FUNCTION_BLOCK PLCopenCommand IMPLEMENTS IPLCopenCommand
VAR
    _PLCopenCommand : PLCopenCommandInternal;
END_VAR

// Copyright (c) 2024 Loupe (https://loupe.team), provided under the MIT License.

IF _PLCopenCommand._status <> PLCopenStatusBase.BUSY AND NOT Execute THEN
    _PLCopenCommand._status := PLCopenStatusBase.NOT_ENABLED;
END_IF

METHOD Aborted : BOOL
VAR_INPUT
END_VAR
// Copyright (c) 2024 Loupe (https://loupe.team), provided under the MIT License.

_PLCopenCommand._status := PLCopenStatusBase.ABORTED;

Remote.Aborted();
Remote := 0;
END_METHOD

METHOD AbortPreviousCommands : BOOL
VAR_INPUT
    newCommand : IPLCopenCommand;
END_VAR
VAR
    i : USINT;
END_VAR
// Copyright (c) 2024 Loupe (https://loupe.team), provided under the MIT License.

//If there is a remote, abort it here
//Don't use this^.abort() because we don't want about ourselves
Remote.Aborted();
Remote := 0;

//Abort any related commands
FOR i := 0 TO GVLTcCommando.MAX_RELATED_GROUPS DO
    IF _PLCopenCommand._commandGroups[i] <> 0 THEN
        _PLCopenCommand._commandGroups[i].AbortPreviousCommands(newCommand);
    END_IF
END_FOR
END_METHOD

METHOD FINAL BaseSize : ULINT
// Copyright (c) 2024 Loupe (https://loupe.team), provided under the MIT License.

BaseSize := SIZEOF(THIS^);
END_METHOD

PROPERTY Consume : BOOL
GET
// Copyright (c) 2024 Loupe (https://loupe.team), provided under the MIT License.

Consume := _PLCopenCommand._Execute;

IF _PLCopenCommand._Execute THEN
    //	THIS^.AbortPreviousCommands( THIS^ );//This is meant to abort if the command comes locally
    _PLCopenCommand._status := PLCopenStatusBase.BUSY;
END_IF

_PLCopenCommand._Execute := FALSE;
END_GET
END_PROPERTY

METHOD Errored : BOOL
VAR_INPUT
    ID : INT;
END_VAR
// Copyright (c) 2024 Loupe (https://loupe.team), provided under the MIT License.

CASE ID OF
    //Any of these statuses are invalid to return as an error.
    //Override to error
    PLCopenStatusBase.BUSY,
        PLCopenStatusBase.ENABLED_WAITING,
        PLCopenStatusBase.ERR_OK:
        _PLCopenCommand._status := PLCopenStatusBase.ERROR;
ELSE
    //Any other status can be passed through
    _PLCopenCommand._status := ID;
END_CASE

Remote.Errored(ID);
END_METHOD

{attribute 'monitoring' := 'call'}
PROPERTY Execute : BOOL
GET
// Copyright (c) 2024 Loupe (https://loupe.team), provided under the MIT License.

Execute := _PLCopenCommand._Execute;
END_GET
SET
// Copyright (c) 2024 Loupe (https://loupe.team), provided under the MIT License.

//We are already executing
IF _PLCopenCommand._Trig = TRUE AND Execute = TRUE THEN

    ; //Do nothing
    //Trigger an execute
ELSIF _PLCopenCommand._Trig = FALSE AND Execute = TRUE THEN
    _PLCopenCommand._status := PLCopenStatusBase.ENABLED_WAITING;
    _PLCopenCommand._Execute := TRUE;

    THIS^.AbortPreviousCommands(THIS^); //This is meant to abort if the command comes locally	

    // We were executing, but resetting it to false;
    // Just resetting execute to false all the time is OK
ELSIF Execute = FALSE THEN
    _PLCopenCommand._Execute := FALSE;
END_IF
END_SET
END_PROPERTY

METHOD FB_init : BOOL
VAR_INPUT
    bInitRetains : BOOL; // if TRUE, the retain variables are initialized (warm start / cold start)
    bInCopyCode : BOOL; // if TRUE, the instance afterwards gets moved into the copy code (online change)
END_VAR
// Copyright (c) 2024 Loupe (https://loupe.team), provided under the MIT License.

_PLCopenCommand._status := PLCopenStatusBase.NOT_ENABLED;
END_METHOD

METHOD Finished : BOOL
VAR_INST
    derived : BOOL;
END_VAR
// Copyright (c) 2024 Loupe (https://loupe.team), provided under the MIT License.

IF _PLCopenCommand._status = PLCopenStatusBase.BUSY THEN
    _PLCopenCommand._status := PLCopenStatusBase.ERR_OK;
END_IF

Remote.Finished();
END_METHOD


METHOD GetSize : ULINT
// Copyright (c) 2024 Loupe (https://loupe.team), provided under the MIT License.

GetSize := SIZEOF(THIS^);
END_METHOD

METHOD GetThis : ULINT
// Copyright (c) 2024 Loupe (https://loupe.team), provided under the MIT License.

GetThis := THIS;
END_METHOD

METHOD RegisterGroup : BOOL
VAR_INPUT
    group : IPLCopenGroup;
END_VAR

VAR
    i : INT;
END_VAR
// Copyright (c) 2024 Loupe (https://loupe.team), provided under the MIT License.

FOR i := 0 TO GVLTcCommando.MAX_RELATED_GROUPS DO
    IF _PLCopenCommand._commandGroups[i] = 0 THEN
        _PLCopenCommand._commandGroups[i] := group;
        EXIT;
    END_IF
END_FOR
END_METHOD

PROPERTY Remote : IPLCopenCall
GET
// Copyright (c) 2024 Loupe (https://loupe.team), provided under the MIT License.

IF _PLCopenCommand._remote <> 0 THEN
    Remote := _PLCopenCommand._remote;
ELSE
    Remote := _PLCopenCommand._nullRemote;
END_IF
END_GET
SET
// Copyright (c) 2024 Loupe (https://loupe.team), provided under the MIT License.

_PLCopenCommand._remote := Remote;
END_SET
END_PROPERTY

{attribute 'monitoring' := 'call'}
PROPERTY Status : PLCopenStatusBase
GET
// Copyright (c) 2024 Loupe (https://loupe.team), provided under the MIT License.

status := _PLCopenCommand._status;
END_GET
END_PROPERTY

END_FUNCTION_BLOCK

(* stored: Version 1.1.0.1
   POU PLCopenCommand: Id {1ef37826-7fac-4345-b9dc-ffeb92b64305}, SpecialFunc None
   Folder API: Id {0587c0fb-5387-4c8e-ab33-b65a12ba1fe4}
   Folder internal: Id {49c08f52-caae-4692-bd2e-016738f72df3}
   Method Aborted: Id {d2af0695-906b-4a1e-be1b-8d6698087918}
   Method AbortPreviousCommands: Id {72a4612a-7755-4ff4-a80f-b8e7a7020c17}
   Method BaseSize: Id {68c25b13-c5d3-4fd8-80c7-c8d81abff00e}
   Property Consume: Id {2ef92d9e-be31-4204-86c4-dd6ebc3c6354}
   Get Get: Id {48f7ff29-f664-4620-8fbe-665cd82855fe}
   Method Errored: Id {e4afdd7d-e3d4-4bb8-9a5c-f28bb8c767d0}
   Property Execute: Id {cf9e92fe-da22-4c8e-b19d-8971f1bd24dd}
   Get Get: Id {15e0faeb-edb9-48e1-b660-f89f647245cb}
   Set Set: Id {a312909e-3f1e-413f-a5a5-82ae3ecc3633}
   Method FB_init: Id {b4349aad-b544-4b1e-a56d-39ff17892797}
   Method Finished: Id {bd7fbae3-272f-4620-a9e2-ef86e3120b6b}
   Method GetSize: Id {6be4e2c5-cb6a-4977-9596-4ad7ba831831}
   Method GetThis: Id {12291a40-cea3-4f5e-bd41-1dabff99abc5}
   Method RegisterGroup: Id {cb5ff1a4-1084-4750-a268-4c2294c40278}
   Property Remote: Id {db1da67f-8a2d-451e-9ac8-181a6de631fa}
   Get Get: Id {144c094c-479d-406d-b7b8-b66e9e7db9d4}
   Set Set: Id {ccf43fee-53f8-4d05-987a-04726b9b683d}
   Property Status: Id {3390b090-03b4-43fa-b62c-451c749fc114}
   Get Get: Id {d49175ec-85a1-4e46-9ed1-546dc054337a} *)
